// Mitsubishi GX Works2 project: codedoan2cuatri   PLC: FX3U/FX3UC

PROGRAM MAIN
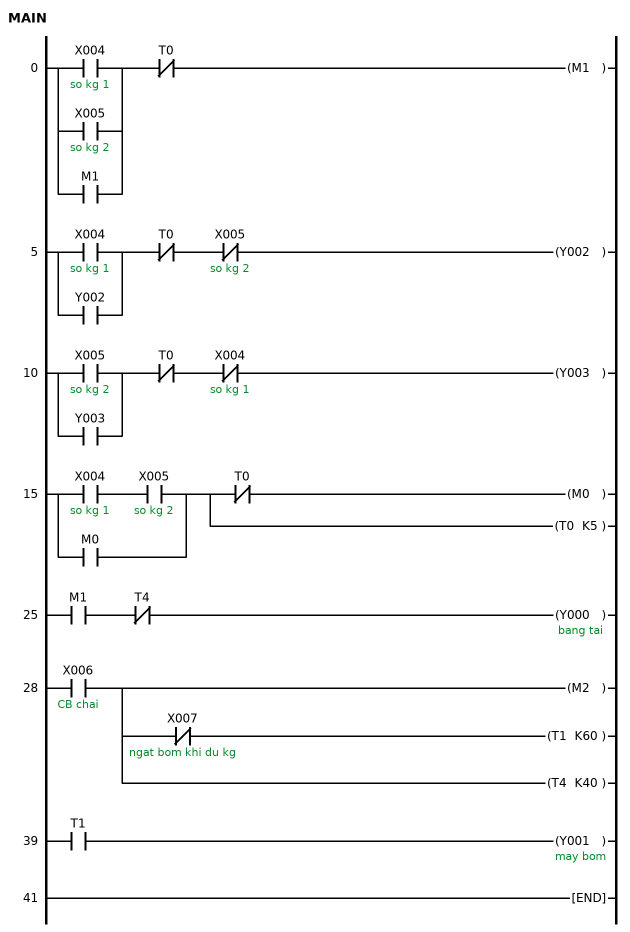
0     LD      X004  ; so kg 1
      OR      X005  ; so kg 2
      OR      M1
      ANI     T0
      OUT     M1
5     LD      X004  ; so kg 1
      OR      Y002
      ANI     T0
      ANI     X005  ; so kg 2
      OUT     Y002
10    LD      X005  ; so kg 2
      OR      Y003
      ANI     T0
      ANI     X004  ; so kg 1
      OUT     Y003
15    LD      X004  ; so kg 1
      AND     X005  ; so kg 2
      OR      M0
      MPS
      ANI     T0
      OUT     M0
      MPP
      OUT     T0 K5
25    LD      M1
      ANI     T4
      OUT     Y000  ; bang tai
28    LD      X006  ; CB chai
      OUT     M2
      MPS
      ANI     X007  ; ngat bom khi du kg
      OUT     T1 K60
      MPP
      OUT     T4 K40
39    LD      T1
      OUT     Y001  ; may bom
41    END
END_PROGRAM
